(*

.. <legal notes>

legal notes
=================
| SPDX-FileCopyrightText: © 2026 Oleksandr Tiutyk <trofimich@gmail.com>
| SPDX-License-Identifier: LGPL-3.0-only
| For details check: LGPL-3.0-only_

.. _LGPL-3.0-only: https://www.gnu.org/licenses/lgpl-3.0.en.html

.. </legal notes>

*)

TYPE AUTOMATION_CONTROLLER_DIAGNOSTICS :
STRUCT
	InitializationError : Core.ERROR;
	
	LastDeviceError : Core.ERROR;
	
	LastWorkingError : Core.ERROR;
	LastStoppingError : Core.ERROR;
	LastFaultError : Core.ERROR;
	
	LastErrorPalce : STRING(39);
END_STRUCT
END_TYPE

(* stored: Version 1.1.0.1
   DUT AUTOMATION_CONTROLLER_DIAGNOSTICS: Id {d49d97a6-34bb-461e-b335-f95dad1f763f} *)
